{attribute 'qualified_only'}
VAR_GLOBAL
	nINTMAXVALUE	: INT := 32767 		; // Integer maximum value 32767
	nINTMINVALUE	: INT := -32767		; // intiger minimum value -32767
	nDINTMAXVALUE	: DINT:= 2147483647 ; // Double integer maximum value 2,147,483,647
	nDINTMINVALUE	: DINT:= -2147483647; // Double integer minimum value -2,147,483,647
END_VAR

(* stored: Version 1.1.0.1, ProductVersion 3.1.4024.4
   GVL GVL_FixedValues: Id {e756683c-0659-42a2-bfb0-c7950b834dce} *)
